// LS Electric XG5000 project: gaze
// PLC LSPLC
// module base 0 slot 0: 입출력 모듈:XBC-DR14E (DC 24V 입력 8점, 릴레이 출력 6점)

PROGRAM NewProgram (task: 스캔 프로그램)

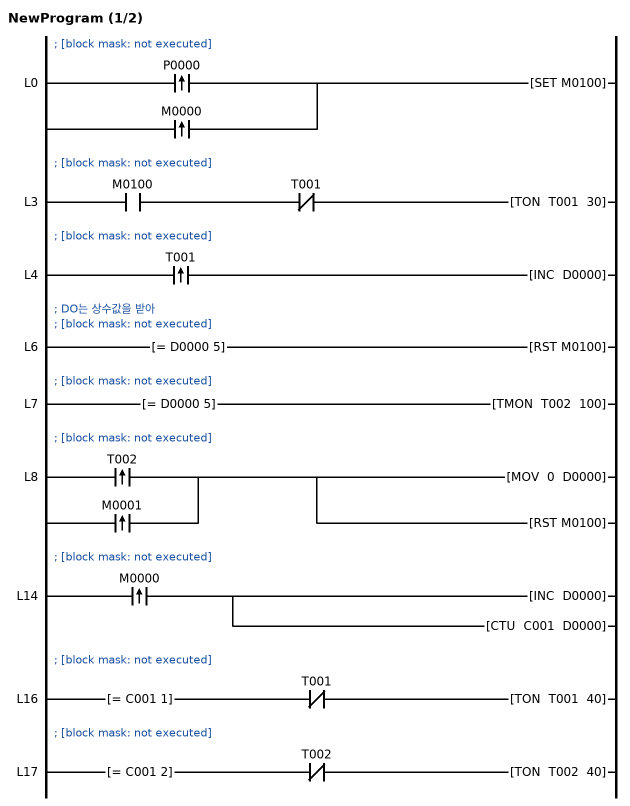
; L0 (block mask: not executed)
LOADP     P0000
ORP       M0000
SET       M0100
; L3 (block mask: not executed)
LOAD      M0100
AND NOT   T001
TON       T001 30
; L4 (block mask: not executed)
LOADP     T001
INC       D0000
// DO는 상수값을 받아
; L6 (block mask: not executed)
LOAD=     D0000 5
RST       M0100
; L7 (block mask: not executed)
LOAD=     D0000 5
TMON      T002 100
; L8 (block mask: not executed)
LOADP     T002
ORP       M0001
MOV       0 D0000
RST       M0100
; L14 (block mask: not executed)
LOADP     M0000
INC       D0000
CTU       C001 D0000
; L16 (block mask: not executed)
LOAD=     C001 1
AND NOT   T001
TON       T001 40
; L17 (block mask: not executed)
LOAD=     C001 2
AND NOT   T002
TON       T002 40

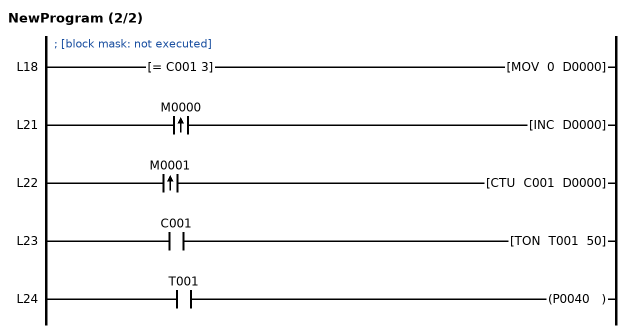
; L18 (block mask: not executed)
LOAD=     C001 3
MOV       0 D0000
; L21
LOADP     M0000
INC       D0000
; L22
LOADP     M0001
CTU       C001 D0000
; L23
LOAD      C001
TON       T001 50
; L24
LOAD      T001
OUT       P0040